ABB RobotStudio station: conveyor CA2.rsstn

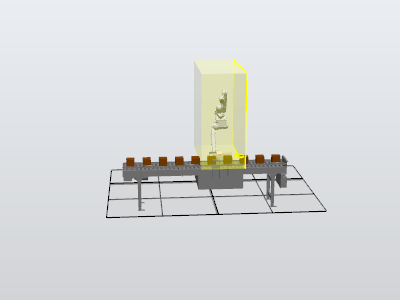
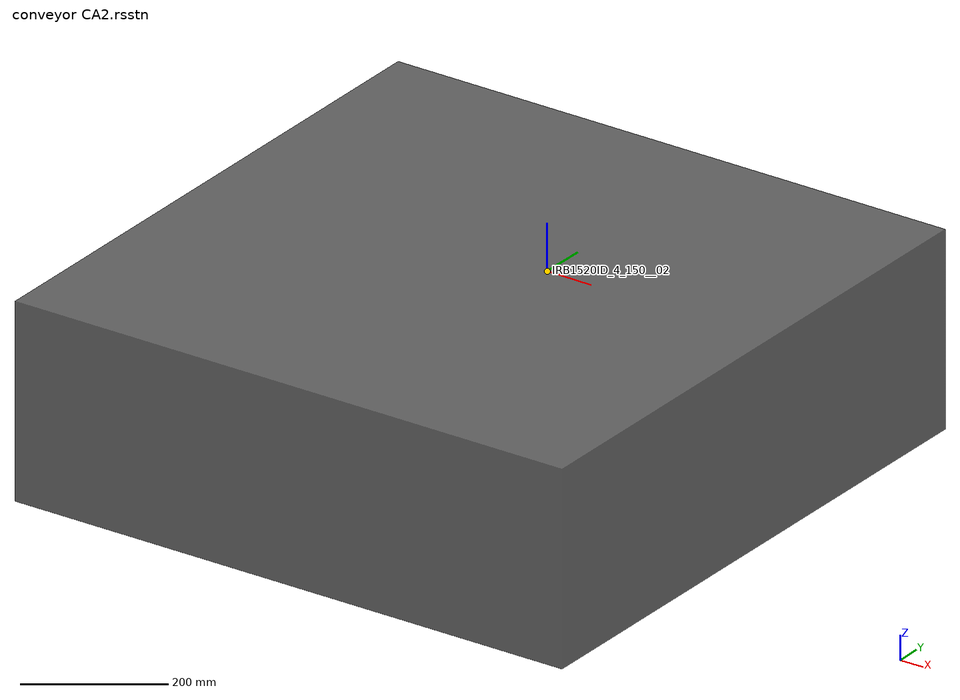
[picture v1: parts stored in the station drawn from their meshes, with robot base, taught points and paths (robot models come from the ABB library and are not in the file)]
Station conveyor (saved by RobotStudio 22.3.10141.1)
Controller Controller21, task T_ROB1: task frame (RAPID world) sits at (-523.8, 1252.27, 775) mm in the station
Controller Controller21
  mechanical unit ROB_1: IRB1520ID_4_150__02, 6 joints, base frame (300, -1000, -553) mm, rotated rx 0 ry 0 rz 90 deg
  mechanical unit CNV1: ?, 1 joints, base frame (0, 0, 0) mm
Layout (positions relative to the parent item):
  - IRB1520ID_4_150__02 [mechanism, from Robots\IRB1520ID_4_150_G_02.rslib] at (-223.8, 252.27, 222) mm, rotated rx 0 ry 0 rz 90 deg; joint values [-0.0349, -0.4346, -0.559, 0.0061, 1.6803, -0.0173] (rad or m)
  - MyTool [mechanism, from Training Objects\myTool.rslib] at (-214.79, 545.25, 1798.38) mm, rotated rx -179.09 ry 50.65 rz -90.37 deg
  - Conveyor [conveyor]
    - 400_guide_2 [part] at (-1298.64, 1249.77, 0) mm, size 3033 x 590 x 945 mm
    - Part_1 [part], size 150 x 150 x 150 mm
    - ConveyorObject_70 [conveyorobject] at (1483.4, 1252.27, 775) mm
      - Part_1 [part] at (0, 100, 0) mm, size 150 x 150 x 150 mm
    - ConveyorObject_71 [conveyorobject] at (1183.4, 1252.27, 775) mm
      - Part_1 [part] at (0, 100, 0) mm, size 150 x 150 x 150 mm
    - ConveyorObject_72 [conveyorobject] at (883.4, 1252.27, 775) mm
      - Part_1 [part] at (0, 100, 0) mm, size 150 x 150 x 150 mm
    - ConveyorObject_73 [conveyorobject] at (583.4, 1252.27, 775) mm
      - Part_1 [part] at (0, 100, 0) mm, size 150 x 150 x 150 mm
    - ConveyorObject_74 [conveyorobject] at (283.4, 1252.27, 775) mm
      - Part_1 [part] at (0, 100, 0) mm, size 150 x 150 x 150 mm
    - ConveyorObject_75 [conveyorobject] at (-16.6, 1252.27, 775) mm
      - Part_1 [part] at (0, 100, 0) mm, size 150 x 150 x 150 mm
    - ConveyorObject_76 [conveyorobject] at (-316.6, 1252.27, 775) mm
      - Part_1 [part] at (0, 100, 0) mm, size 150 x 150 x 150 mm
    - ConveyorObject_12 [conveyorobject] at (-616.6, 1252.27, 775) mm
      - Part_1 [part] at (0, 100, 0) mm, size 150 x 150 x 150 mm
    - ConveyorObject_13 [conveyorobject] at (-916.6, 1252.27, 775) mm
      - Part_1 [part] at (0, 100, 0) mm, size 150 x 150 x 150 mm
    - ConveyorObject_11 [conveyorobject] at (-1216.6, 1252.27, 775) mm
      - Part_1 [part] at (0, 100, 0) mm, size 150 x 150 x 150 mm
  - SmartComponent_1 [smart component]
  - Group_1 [graphiccomponentgroup]
  - Part_3 [part] at (-667.24, -364.74, 0) mm, size 900 x 900 x 300 mm
Attachment: MyTool is attached to IRB1520ID_4_150__02 / Link6
Conveyor tracking Connection: unit CNV1, TravelOffset=0.7, QueueTrackDistance=0, StartWindowWidth=0.8, SyncSeparation=0.1, CountsPerMeter=10000
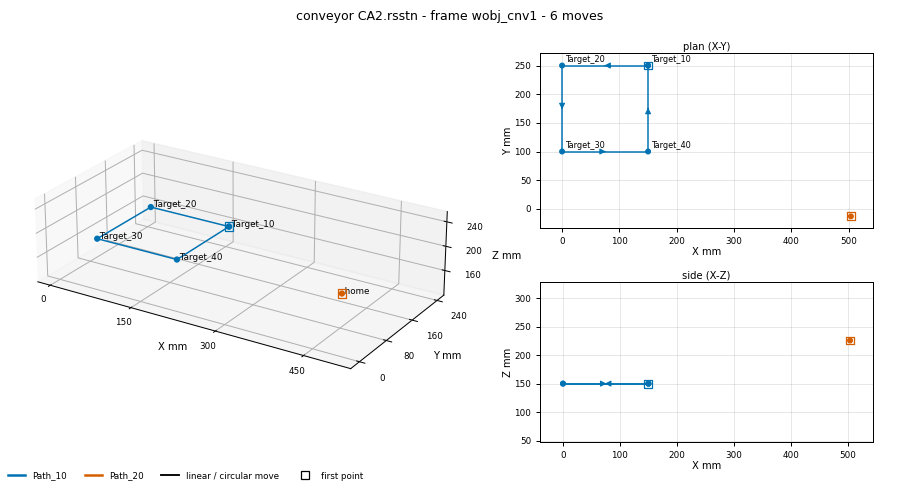
[picture p0: tool path of conveyor CA2.rsstn in frame wobj_cnv1, 6 of 6 moves have a stored position in this frame; points joined in program order, loops and branches not executed]
Targets, tools, work objects and paths stored in the station, written as RAPID:
! task T_ROB1
MODULE CalibData
  PERS tooldata MyTool:=[TRUE,[[31.792631019,0,229.638935148],[0.945518576,0,0.325568154,0]],[1,[0,0,1],[1,0,0,0],0,0,0]];
  TASK PERS wobjdata wobj_cnv1:=[FALSE,FALSE,"CNV1",[[0,0,0],[1,0,0,0]],[[0,0,0],[1,0,0,0]]];
ENDMODULE

! task T_ROB1
MODULE Module1
  CONST robtarget home:=[[503.789233124,-13.084410881,225.64730631],[0.134922335,-0.694115238,0.694115238,0.134922335],[0,0,0,0],[9E+09,9E+09,9E+09,9E+09,9E+09,0]];
  CONST robtarget Target_10:=[[150.000012703,249.999784325,149.999988896],[0.134921848,-0.694115329,0.694115327,0.134921895],[0,-1,0,0],[9E+09,9E+09,9E+09,9E+09,9E+09,0]];
  CONST robtarget Target_20:=[[0.000016939,249.999781564,149.999991428],[0.134921717,-0.694115356,0.69411535,0.134921768],[0,-1,0,0],[9E+09,9E+09,9E+09,9E+09,9E+09,0]];
  CONST robtarget Target_30:=[[0.000045139,99.999676408,150.000015376],[0.134921665,-0.694115373,0.694115358,0.13492169],[0,-1,0,0],[9E+09,9E+09,9E+09,9E+09,9E+09,0]];
  CONST robtarget Target_40:=[[150.000027473,99.999674464,149.999995787],[0.134921678,-0.694115381,0.694115356,0.134921653],[0,-1,0,0],[9E+09,9E+09,9E+09,9E+09,9E+09,0]];
  PROC Path_10()
    MoveL Target_10,v1000,fine,MyTool\WObj:=wobj_cnv1;
    MoveL Target_20,v1000,fine,MyTool\WObj:=wobj_cnv1;
    MoveL Target_30,v1000,fine,MyTool\WObj:=wobj_cnv1;
    MoveL Target_40,v1000,fine,MyTool\WObj:=wobj_cnv1;
    MoveL Target_10,v1000,fine,MyTool\WObj:=wobj_cnv1;
  ENDPROC
  PROC Path_20()
    MoveL home,v1000,z100,MyTool\WObj:=wobj_cnv1;
    ActUnit CNV1;
    WaitWObj wobj_cnv1;
    Path_10;
    WaitWObj wobj_cnv1;
  ENDPROC
ENDMODULE

